ABB RobotStudio station: Lab2.rspag

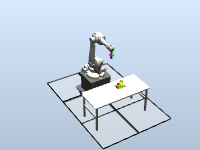
--- station ---
Station Lab2 (saved by RobotStudio 6.8.8307.1040)
Controller System1, task T_ROB1: task frame (RAPID world) sits at (0, 0, 520) mm in the station
Controller System1
  mechanical unit ROB_1: IRB1600_10_145__01, 6 joints, base frame (0, 0, 0) mm
Layout (positions relative to the parent item):
  - IRB1600_10_145__01 [mechanism, from Robots\IRB1600_10_145_G_01.rslib] at (0, 0, 520) mm; joint values [0, 0, 0, 0, 1.5708, 0] (rad or m)
  - pen [mechanism, from Libraries\pen.rslib] at (750, 0, 1641.5) mm, rotated rx 180 ry 0 rz 180 deg
  - table_for_robot [part, from Libraries\table_for_robot.rslib]
  - work_table [part, from Libraries\work_table.rslib] at (800, -800, 0) mm, rotated rx 0 ry 0 rz 90 deg
Attachment: pen is attached to IRB1600_10_145__01 / Link6

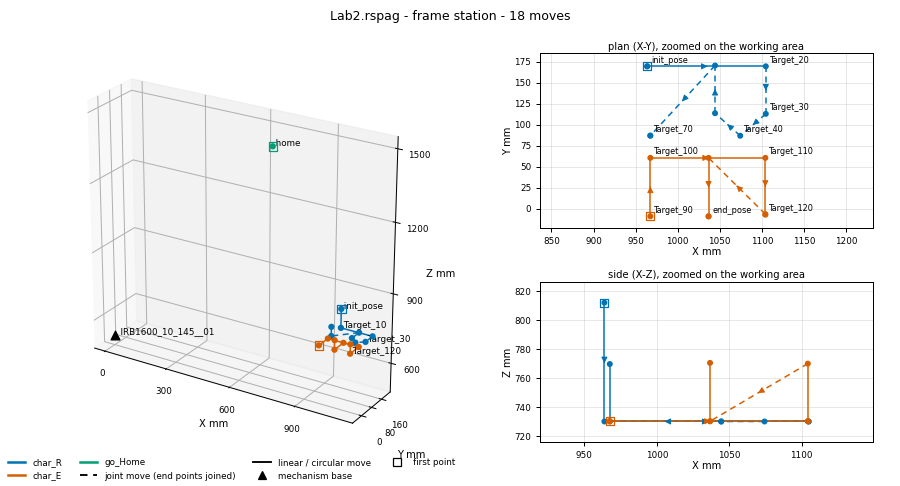
[picture p0: tool path of Lab2.rspag in frame station, 18 of 18 moves have a stored position in this frame; points joined in program order, loops and branches not executed]
--- Backups/System1/RAPID/TASK1/PROGMOD/CalibData.mod ---
MODULE CalibData
	PERS tooldata pen:=[TRUE,[[0,0,139],[1,0,0,0]],[0.5,[0,0,20],[1,0,0,0],0,0,0]];
	TASK PERS wobjdata wobjTable:=[FALSE,TRUE,"",[[747.33,-871.732,210.071],[1,0,0,0]],[[0,0,0],[1,0,0,0]]];
ENDMODULE

--- Backups/System1/RAPID/TASK1/PROGMOD/Module1.mod ---
MODULE Module1
	CONST robtarget init_pose:=[[216.461714459,1041.265991727,81.999249998],[-0.000000071,-0.000000006,1,-0.000000022],[0,-1,0,0],[9E+09,9E+09,9E+09,9E+09,9E+09,9E+09]];
	CONST robtarget Target_10:=[[216.461718177,1041.265992381,-0.039384878],[-0.000000071,-0.000000002,1,-0.000000022],[0,-1,0,0],[9E+09,9E+09,9E+09,9E+09,9E+09,9E+09]];
	CONST robtarget Target_20:=[[357.448040772,1041.266003704,-0.039371256],[-0.000000072,-0.000000006,1,-0.000000022],[0,-1,0,0],[9E+09,9E+09,9E+09,9E+09,9E+09,9E+09]];
	CONST robtarget Target_30:=[[357.448046402,984.74128717,-0.039363275],[-0.000000057,-0.000000003,1,-0.000000021],[0,-1,0,0],[9E+09,9E+09,9E+09,9E+09,9E+09,9E+09]];
	CONST robtarget Target_40:=[[327.012967805,958.724705453,-0.03934658],[-0.000000036,-0.000000006,1,-0.000000019],[0,-1,0,0],[9E+09,9E+09,9E+09,9E+09,9E+09,9E+09]];
	CONST robtarget Target_50:=[[297.113959914,985.511099362,-0.03927025],[-0.000000067,-0.000000005,1,-0.000000021],[0,-1,0,0],[9E+09,9E+09,9E+09,9E+09,9E+09,9E+09]];
	CONST robtarget Target_60:=[[297.113959919,1042.1893038,-0.03926682],[-0.000000055,-0.000000007,1,-0.000000019],[0,-1,0,0],[9E+09,9E+09,9E+09,9E+09,9E+09,9E+09]];
	CONST robtarget Target_70:=[[220.193685145,958.869251733,-0.039269098],[-0.000000043,-0.000000008,1,-0.000000018],[0,-1,0,0],[9E+09,9E+09,9E+09,9E+09,9E+09,9E+09]];
	CONST robtarget Target_80:=[[220.193690021,958.869252172,39.627339114],[-0.000000035,-0.000000009,1,-0.000000018],[0,-1,0,0],[9E+09,9E+09,9E+09,9E+09,9E+09,9E+09]];
	CONST robtarget Target_90:=[[220.19369359,863.027556433,0.148656861],[-0.000000022,-0.00000001,1,-0.000000018],[-1,-1,-1,0],[9E+09,9E+09,9E+09,9E+09,9E+09,9E+09]];
	CONST robtarget Target_100:=[[220.193689256,932.458171989,0.148743709],[-0.000000013,-0.000000012,1,-0.000000017],[0,-1,0,0],[9E+09,9E+09,9E+09,9E+09,9E+09,9E+09]];
	CONST robtarget Target_110:=[[356.895981016,932.45816693,0.148727049],[-0.000000021,-0.000000011,1,-0.000000018],[0,-1,0,0],[9E+09,9E+09,9E+09,9E+09,9E+09,9E+09]];
	CONST robtarget Target_120:=[[356.895968626,864.911696335,0.148697911],[-0.000000052,-0.000000011,1,-0.000000018],[-1,-1,-1,0],[9E+09,9E+09,9E+09,9E+09,9E+09,9E+09]];
	CONST robtarget Target_130:=[[356.895982834,865.541145089,39.914148887],[-0.000000018,-0.000000011,1,-0.000000018],[-1,-1,-1,0],[9E+09,9E+09,9E+09,9E+09,9E+09,9E+09]];
	CONST robtarget Target_140:=[[289.395030822,932.471849734,0.117301704],[-0.000000054,-0.000000011,1,-0.000000019],[0,-1,0,0],[9E+09,9E+09,9E+09,9E+09,9E+09,9E+09]];
	CONST robtarget Target_150:=[[289.395036619,862.943540985,0.117327628],[-0.000000048,-0.000000011,1,-0.000000019],[-1,-1,-1,0],[9E+09,9E+09,9E+09,9E+09,9E+09,9E+09]];
	CONST robtarget end_pose:=[[289.395029601,862.943541045,40.413119991],[-0.000000056,-0.000000011,1,-0.000000019],[-1,-1,-1,0],[9E+09,9E+09,9E+09,9E+09,9E+09,9E+09]];
	CONST robtarget home:=[[750,0,982.5],[0,0,1,0],[0,0,0,0],[9E+09,9E+09,9E+09,9E+09,9E+09,9E+09]];
    !***********************************************************
    !
    ! Module:  Module1
    !
    ! Description:
    !   <Insert description here>
    !
    ! Author: R. Eidelman
    !
    ! Version: 1.0
    !
    !***********************************************************


    !***********************************************************
    !
    ! Procedure main
    !
    !   This is the entry point of your program
    !
    !***********************************************************
    PROC main()
		go_Home;
		char_R;
		char_E;
		go_Home;
        !Add your code here
    ENDPROC
	PROC char_R()
	    MoveJ init_pose,v100,fine,pen\WObj:=wobjTable;
	    MoveL Target_10,v100,fine,pen\WObj:=wobjTable;
	    MoveL Target_20,v100,fine,pen\WObj:=wobjTable;
	    MoveJ Target_30,v100,z30,pen\WObj:=wobjTable;
	    MoveJ Target_40,v100,z100,pen\WObj:=wobjTable;
	    MoveJ Target_50,v100,z40,pen\WObj:=wobjTable;
	    MoveJ Target_60,v100,fine,pen\WObj:=wobjTable;
	    MoveJ Target_70,v100,fine,pen\WObj:=wobjTable;
	    MoveL Target_80,v100,fine,pen\WObj:=wobjTable;
	ENDPROC
	PROC char_E()
	    MoveJ Target_90,v100,fine,pen\WObj:=wobjTable;
	    MoveL Target_100,v100,fine,pen\WObj:=wobjTable;
	    MoveL Target_110,v100,fine,pen\WObj:=wobjTable;
	    MoveL Target_120,v100,fine,pen\WObj:=wobjTable;
	    MoveL Target_130,v100,fine,pen\WObj:=wobjTable;
	    MoveJ Target_140,v100,fine,pen\WObj:=wobjTable;
	    MoveL Target_150,v100,fine,pen\WObj:=wobjTable;
	    MoveL end_pose,v100,fine,pen\WObj:=wobjTable;
	ENDPROC
	PROC go_Home()
	    MoveJ home,v100,fine,pen\WObj:=wobj0;
	ENDPROC
ENDMODULE
